// Mitsubishi GX Works2 project: 세탁기   PLC: Q03UDV

PROGRAM MAIN
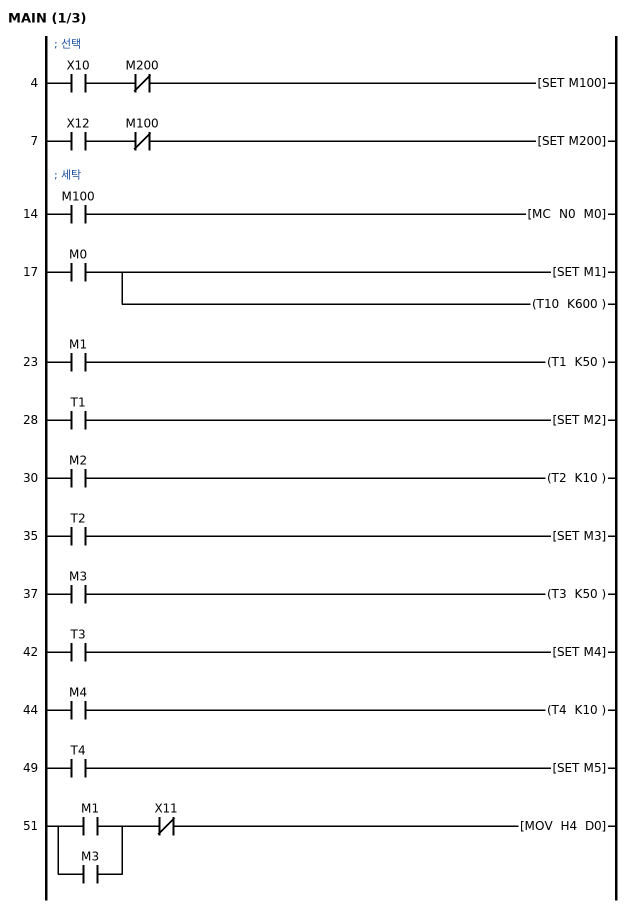
; 선택
4     LD      X10
      ANI     M200
      SET     M100
7     LD      X12
      ANI     M100
      SET     M200
; 세탁
14    LD      M100
      MC      N0 M0
17    LD      M0
      SET     M1
      OUT     T10 K600
23    LD      M1
      OUT     T1 K50
28    LD      T1
      SET     M2
30    LD      M2
      OUT     T2 K10
35    LD      T2
      SET     M3
37    LD      M3
      OUT     T3 K50
42    LD      T3
      SET     M4
44    LD      M4
      OUT     T4 K10
49    LD      T4
      SET     M5
51    LD      M1
      OR      M3
      ANI     X11
      MOV     H4 D0
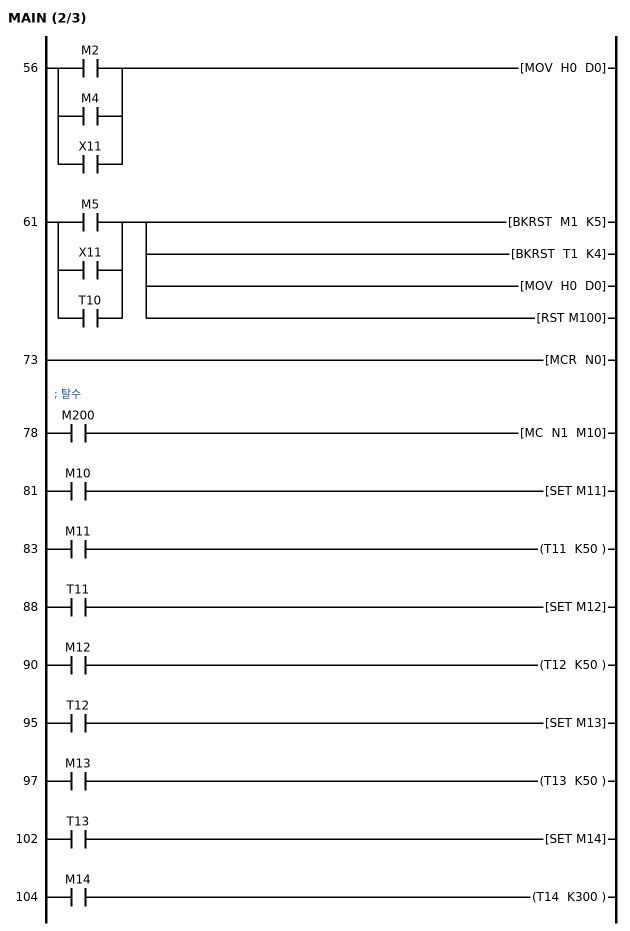
56    LD      M2
      OR      M4
      OR      X11
      MOV     H0 D0
61    LD      M5
      OR      X11
      OR      T10
      BKRST   M1 K5
      BKRST   T1 K4
      MOV     H0 D0
      RST     M100
73    MCR     N0
; 탈수
78    LD      M200
      MC      N1 M10
81    LD      M10
      SET     M11
83    LD      M11
      OUT     T11 K50
88    LD      T11
      SET     M12
90    LD      M12
      OUT     T12 K50
95    LD      T12
      SET     M13
97    LD      M13
      OUT     T13 K50
102   LD      T13
      SET     M14
104   LD      M14
      OUT     T14 K300
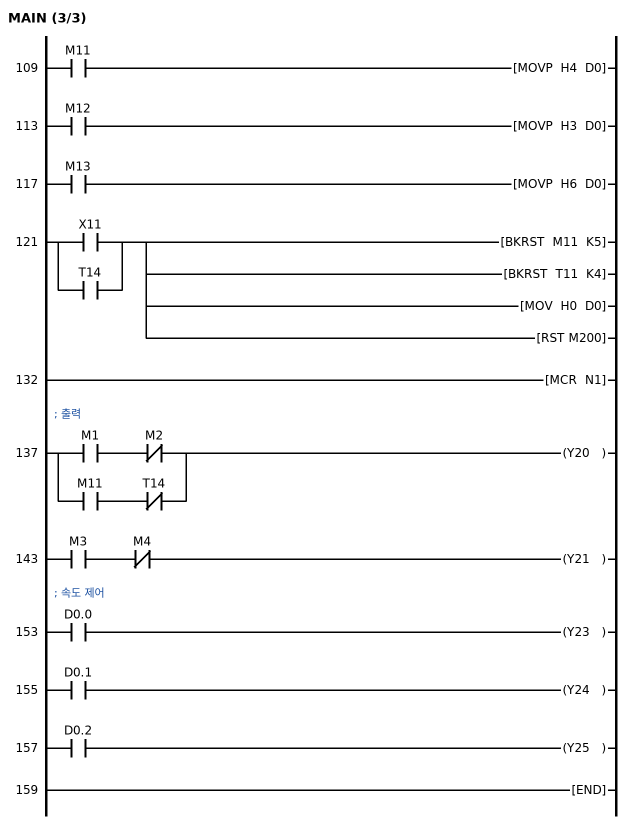
109   LD      M11
      MOVP    H4 D0
113   LD      M12
      MOVP    H3 D0
117   LD      M13
      MOVP    H6 D0
121   LD      X11
      OR      T14
      BKRST   M11 K5
      BKRST   T11 K4
      MOV     H0 D0
      RST     M200
132   MCR     N1
; 출력
137   LD      M1
      ANI     M2
      LD      M11
      ANI     T14
      ORB
      OUT     Y20
143   LD      M3
      ANI     M4
      OUT     Y21
; 속도 제어
153   LD      D0.0
      OUT     Y23
155   LD      D0.1
      OUT     Y24
157   LD      D0.2
      OUT     Y25
159   END
END_PROGRAM

PROGRAM MAIN1
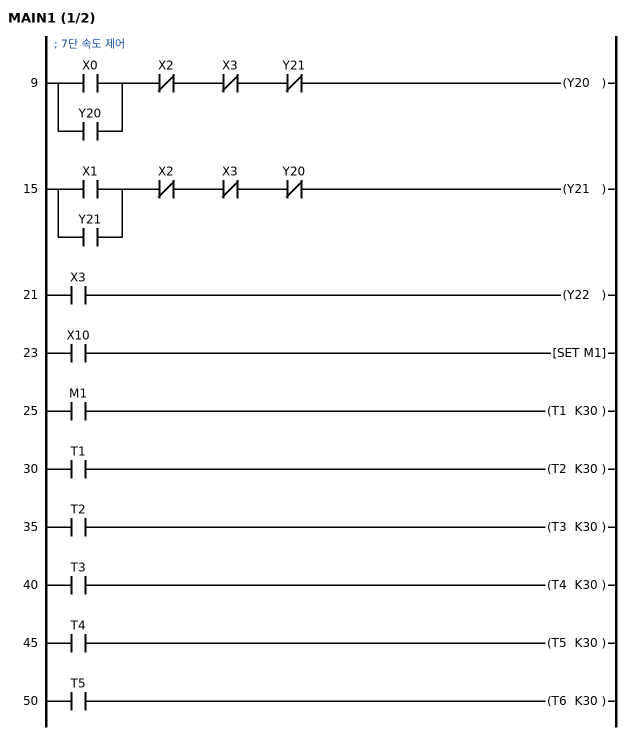
; 7단 속도 제어
9     LD      X0
      OR      Y20
      ANI     X2
      ANI     X3
      ANI     Y21
      OUT     Y20
15    LD      X1
      OR      Y21
      ANI     X2
      ANI     X3
      ANI     Y20
      OUT     Y21
21    LD      X3
      OUT     Y22
23    LD      X10
      SET     M1
25    LD      M1
      OUT     T1 K30
30    LD      T1
      OUT     T2 K30
35    LD      T2
      OUT     T3 K30
40    LD      T3
      OUT     T4 K30
45    LD      T4
      OUT     T5 K30
50    LD      T5
      OUT     T6 K30
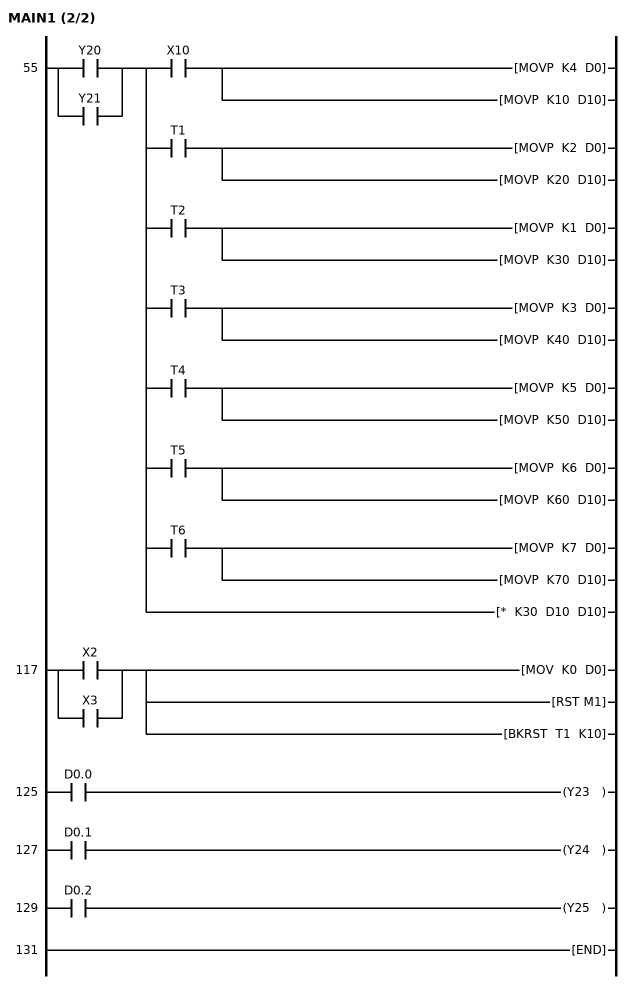
55    LD      Y20
      OR      Y21
      MPS
      AND     X10
      MOVP    K4 D0
      MOVP    K10 D10
      MRD
      AND     T1
      MOVP    K2 D0
      MOVP    K20 D10
      MRD
      AND     T2
      MOVP    K1 D0
      MOVP    K30 D10
      MRD
      AND     T3
      MOVP    K3 D0
      MOVP    K40 D10
      MRD
      AND     T4
      MOVP    K5 D0
      MOVP    K50 D10
      MRD
      AND     T5
      MOVP    K6 D0
      MOVP    K60 D10
      MRD
      AND     T6
      MOVP    K7 D0
      MOVP    K70 D10
      MPP
      *       K30 D10 D10
117   LD      X2
      OR      X3
      MOV     K0 D0
      RST     M1
      BKRST   T1 K10
125   LD      D0.0
      OUT     Y23
127   LD      D0.1
      OUT     Y24
129   LD      D0.2
      OUT     Y25
131   END
END_PROGRAM
